// TIA Portal V20 export
TYPE "LBP_typeMcp483TurningOutput"
TITLE = MCP 483 image / Image du MCP 483
// Output image of MCP 483 Turning / Image de sortie du MCP 483 Tournage
   STRUCT
      auto : Bool;
      mda : Bool;
      teachIn : Bool;
      jog : Bool;
      inc1 : Bool;
      inc10 : Bool;
      inc100 : Bool;
      inc1000 : Bool;
      inc10000 : Bool;
      incVar : Bool;
      refPoint : Bool;
      repos : Bool;
      cycleStop : Bool;
      cycleStart : Bool;
      feedrateStop : Bool;
      feedrateStart : Bool;
      spindleStop : Bool;
      spindleStart : Bool;
      singleBlock : Bool;
      r10 : Bool;   // R10
      axisCMinus : Bool;   // R7
      axisZMinus : Bool;   // R4
      axisYPlus : Bool;   // R1
      r13 : Bool;   // R13
      r15 : Bool;   // R15
      axisZPlus : Bool;   // R6
      axisXMinus : Bool;   // R8
      axisYMinus : Bool;   // R9
      r11 : Bool;   // R11
      mcsWcs : Bool;   // R12
      rapidTraverse : Bool;   // R5
      axisCPlus : Bool;   // R3
      axisXPlus : Bool;   // R2
      customerKey15 : Bool;   // T15
      customerKey14 : Bool;   // T14
      customerKey13 : Bool;   // T13
      customerKey12 : Bool;   // T12
      customerKey11 : Bool;   // T11
      customerKey10 : Bool;   // T10
      customerKey9 : Bool;   // T9
      customerKey8 : Bool;   // T8
      customerKey7 : Bool;   // T7
      customerKey6 : Bool;   // T6
      customerKey5 : Bool;   // T5
      customerKey4 : Bool;   // T4
      customerKey3 : Bool;   // T3
      customerKey2 : Bool;   // T2
      customerKey1 : Bool;   // T1
   END_STRUCT;
END_TYPE
